TYPE CmpConvBreakStopGroup :
STRUCT
	Framework: Framework;
	ConvRunning: ARRAY[1..cBreakStopGroupMaxInstance] OF BOOL;
	LowerStopReq: ARRAY[1..cBreakStopGroupMaxInstance] OF BOOL;
	Config: CmpConvBreakStopGroupConfig;
END_STRUCT
END_TYPE

(* stored: Version 1.1.0.1, ProductVersion 3.1.4024.6
   DUT CmpConvBreakStopGroup: Id {12a464f6-193e-4ceb-a9eb-f57d288f209b} *)
